// Mitsubishi GX Works2 project: Tap2V2FX3U   PLC: FX3U/FX3UC

// global labels: Global1
VAR_GLOBAL
  XXLimitN AT M8344 : BOOL;
  XXLimitP AT M8343 : BOOL;
  XXBusy AT M8340 : BOOL;
  XXInterruptInverse AT M8347 : BOOL;
  XXPos AT D8340 : DINT;
  XXAccelTime AT D8348 : INT;
  XXDecelTime AT D8349 : INT;
  XXPosView AT D0 : DINT;
  XXTarPos AT D2 : DINT;
  XXFeed AT D4 : DINT;
  XXPPR AT D6 : DINT;
  XXTarR AT M0 : BOOL;
  XXTarRSkip AT D8 : INT;
  XXOn AT M1 : BOOL;
  XXRun AT M2 : BOOL;
  XXDirection AT M3 : BOOL;
  XXMinI AT X000 : BOOL;
  XXReady AT M4 : BOOL;
  XXReadyI AT X004 : BOOL;
  XXPulseO AT Y000 : BOOL;
  XXDirectionO AT Y004 : BOOL;
  XXOnO AT Y010 : BOOL;
  XXInTorqueI AT X010 : BOOL;
  XXInTorqueIEdge AT M5 : BOOL;
  XXOverTorque AT M6 : BOOL;
  YYLimitN AT M8354 : BOOL;
  YYLimitP AT M8353 : BOOL;
  YYBusy AT M8350 : BOOL;
  YYInterruptInverse AT M8357 : BOOL;
  YYPos AT D8350 : DINT;
  YYAccelTime AT D8358 : INT;
  YYDecelTime AT D8359 : INT;
  YYPosView AT D9 : DINT;
  YYTarPos AT D11 : DINT;
  YYFeed AT D13 : DINT;
  YYPPM AT D15 : DINT;
  YYTarR AT M7 : BOOL;
  YYTarRSkip AT D17 : INT;
  YYOn AT M8 : BOOL;
  YYRun AT M9 : BOOL;
  YYDirection AT M10 : BOOL;
  YYReady AT M11 : BOOL;
  YYReadyI AT X005 : BOOL;
  YYPulseO AT Y001 : BOOL;
  YYDirectionO AT Y005 : BOOL;
  YYOnO AT Y011 : BOOL;
  YYInTorqueI AT X011 : BOOL;
  YYInTorqueIEdge AT M12 : BOOL;
  YYOverTorque AT M13 : BOOL;
  ZZLimitN AT M8364 : BOOL;
  ZZLimitP AT M8363 : BOOL;
  ZZBusy AT M8360 : BOOL;
  ZZInterruptInverse AT M8367 : BOOL;
  ZZPos AT D8360 : DINT;
  ZZAccelTime AT D8368 : INT;
  ZZDecelTime AT D8369 : INT;
  ZZPosView AT D18 : DINT;
  ZZTarPos AT D20 : DINT;
  ZZFeed AT D22 : DINT;
  ZZPPR AT D24 : DINT;
  ZZTarR AT M14 : BOOL;
  ZZTarRSkip AT D26 : INT;
  ZZRun AT M15 : BOOL;
  ZZDirection AT M16 : BOOL;
  ZZReadyI AT X006 : BOOL;
  ZZPulseO AT Y002 : BOOL;
  ZZDirectionO AT Y006 : BOOL;
  ZZOnO AT Y012 : BOOL;
  ZZInTorqueI AT X012 : BOOL;
  ZZInTorqueIEdge AT M17 : BOOL;
  ZZOverTorque AT M18 : BOOL;
  RunState AT D27 : INT;
  RunStateNext AT M19 : BOOL;
  AxisSpinState AT D28 : INT;
  AxisSpinStateNext AT M20 : BOOL;
  AxisTapState AT D29 : INT;
  AxisTapStateNext AT M21 : BOOL;
  FoilExtractState AT D30 : INT;
  FoilExtractStateNext AT M22 : BOOL;
  FoilClampState AT D31 : INT;
  FoilClampStateNext AT M23 : BOOL;
  FoilSupplyState AT D32 : INT;
  FoilSupplyStateNext AT M24 : BOOL;
  FoilExtractDropN AT M25 : BOOL;
  FoilExtractDropNTimer AT TC0 : BOOL;
  FoilExtractDropNTimerDelay AT D33 : INT;
  FoilExtractDropP AT M26 : BOOL;
  FoilExtractDropPTimer AT TC1 : BOOL;
  FoilExtractDropPTimerDelay AT D34 : INT;
  FoilExtractDrop AT M27 : BOOL;
  FoilExtractDropO AT Y003 : BOOL;
  FoilClampN AT M28 : BOOL;
  FoilClampNTimer AT TC2 : BOOL;
  FoilClampNTimerDelay AT D35 : INT;
  FoilClampP AT M29 : BOOL;
  FoilClampPTimer AT TC3 : BOOL;
  FoilClampPTimerDelay AT D36 : INT;
  FoilClampPI AT X001 : BOOL;
  FoilClamp AT M30 : BOOL;
  FoilClampO AT Y007 : BOOL;
  FoilSupply AT M31 : BOOL;
  FoilSupplyO AT Y013 : BOOL;
  WorkFeedSpin AT D37 : DINT;
  WorkFeedTapTravelFast AT D39 : DINT;
  WorkFeedTapSpinDown AT D41 : DINT;
  WorkFeedTapSpinUp AT D43 : DINT;
  FoilFull AT M32 : BOOL;
  FoilFullI AT X002 : BOOL;
  FoilFullTimer AT TC4 : BOOL;
  SpinArray AT D45 : ARRAY [0..7] OF DINT;
  SpinArrayIndex AT D61 : INT;
  AirReady AT M33 : BOOL;
  AirReadyI AT X003 : BOOL;
  Run AT M34 : BOOL;
  RunI AT X007 : BOOL;
  RunStop AT M35 : BOOL;
  RunStopI AT X013 : BOOL;
  SettingTapPitch AT D62 : DINT;
  SettingTapPitchI AT X014 : BOOL;
  SettingFoilSupplyI AT X015 : BOOL;
  SettingTapSpinSpeedI AT X016 : BOOL;
  SettingTapTravelLengthIObsolete AT X017 : BOOL;
  SettingTapTravelBegin AT D64 : DINT;
  SettingTapTravelBeginOffset AT D66 : DINT;
  SettingTapTravelFast AT D68 : DINT;
  SettingTapTravelEnd AT D70 : DINT;
  TapMoveToTravelBegin AT M36 : BOOL;
  TapCount AT D72 : DINT;
  TapCountAtSupplyEnd AT D74 : DINT;
  TapCountResetOrigin AT D76 : DINT;
  StopTap AT M37 : BOOL;
  StopTapTimer AT TC5 : BOOL;
  StopClamp AT M38 : BOOL;
  StopClampPLS AT M39 : BOOL;
  StopClampTimer AT TC6 : BOOL;
  XXOff AT M40 : BOOL;
  XXOffTimer AT TC7 : BOOL;
  Alert AT M41 : BOOL;
  AlertTimer AT TC8 : BOOL;
  AlertO AT Y014 : BOOL;
  ErrorReset AT M42 : BOOL;
  ErrorResetTimer AT TC9 : BOOL;
  ErrorResetO AT Y015 : BOOL;
  OverloadTimer AT TC256 : BOOL;
  OverloadTimerEN AT M43 : BOOL;
  Overload AT M44 : BOOL;
  SettingTapPitchBoolCounter1000 AT D78 : INT;
  SettingTapPitchBoolCounter1270 AT D79 : INT;
  SettingTapPitchBool AT M45 : BOOL;
  SettingTapPitchBoolO AT Y016 : BOOL;
  SettingTapPitchDone AT M46 : BOOL;
END_VAR

// task Task_01 (event TRUE, interval 0, priority 31): POU_01

PROGRAM POU_01
VAR
  fTmp : BOOL;
  fSpace : DINT;
  fCount : INT;
  fNeedResetOrigin : BOOL;
END_VAR
SET(M8002, M8336);
MOV(M8002, HFFF0, D8336);
RST(M8002, XXInterruptInverse);
RST(M8002, XXOn);
RST(M8002, YYOn);
MOV(M8002, 50, XXAccelTime);
MOV(M8002, 50, XXDecelTime);
MOV(M8002, 250, YYAccelTime); MOV(M8002, YYAccelTime, ZZAccelTime);
MOV(M8002, 250, YYDecelTime); MOV(M8002, YYDecelTime, ZZDecelTime);
RST(M8002, XXOverTorque);
RST(M8002, YYOverTorque);
RST(M8002, ZZOverTorque);
RST(M8002, FoilExtractDrop);
RST(M8002, FoilClamp);
RST(M8002, FoilSupply);
SET(M8002, Alert);
(*x axis: index spin*)
DMOV(M8002, 131_072, XXPPR);
MOV(M8002, 8, fCount);
DMOV(M8002, XXPPR / INT_TO_DINT(fCount), fSpace);
DMOV(M8002, fSpace * 0, SpinArray[0]);
DMOV(M8002, fSpace * 1, SpinArray[1]);
DMOV(M8002, fSpace * 2, SpinArray[2]);
DMOV(M8002, fSpace * 3, SpinArray[3]);
DMOV(M8002, fSpace * 4, SpinArray[4]);
DMOV(M8002, fSpace * 5, SpinArray[5]);
DMOV(M8002, fSpace * 6, SpinArray[6]);
DMOV(M8002, fSpace * 7, SpinArray[7]);
DMOV(M8002, 98_304, WorkFeedSpin);
(*y axis: tap travel*)
DMOV(M8002, 1_000, YYPPM);
RST(M8002, TapCount);
DMOV(M8002, 100_000, WorkFeedTapTravelFast);
(*z axis: tap spin*)
DMOV(M8002, YYPPM, ZZPPR);
(*it easier to calculate if YYPPM = ZZPPR*)
(*|||||||||||||||*)

(*|||||||||||||||*)
SET(Run AND RunState = 0 AND AirReady AND SettingTapPitchDone, fTmp);
RST(fTmp, Run);
SET(fTmp, XXOn);
SET(fTmp, YYOn);
SET(fTmp, TapMoveToTravelBegin);
RST(fTmp, StopClamp);
MOV(fTmp, 1, RunState);
RST(fTmp, fTmp);
SET(RunStop OR Overload, fTmp);
SET(fTmp AND RunStop, ErrorReset);
RST(fTmp, Run);
RST(fTmp, RunStop);
RST(fTmp, Overload);
SET(fTmp, Alert);
ZRST(fTmp, RunState, FoilSupplyState);
RST(fTmp, XXRun);
RST(fTmp, XXOn);
RST(fTmp, YYRun);
RST(fTmp, ZZRun);
SET(fTmp AND YYOn, StopTap);
RST(fTmp, FoilExtractDrop);
RST(fTmp, FoilClamp);
RST(fTmp, FoilSupply);
RST(fTmp, fTmp);
OUT_T(StopTap, StopTapTimer, 5);
RST(StopTapTimer, YYOn);
RST(StopTapTimer, StopTap);

(*|||||||||||||||*)
(*|||||||||||||||*)
INC(RunStateNext, RunState);
INC(AxisSpinStateNext, AxisSpinState);
INC(AxisTapStateNext, AxisTapState);
INC(FoilExtractStateNext, FoilExtractState);
INC(FoilClampStateNext, FoilClampState);
INC(FoilSupplyStateNext, FoilSupplyState);
ZRST(M8000, RunStateNext, FoilSupplyStateNext);
DECO(M8000, RunState, 6, M100);
DECO(M8000, AxisSpinState, 6, M200); DECO(M8000, AxisSpinState, 6, M1200); ZRST(NOT XXReady, M1200, M1263);
DECO(M8000, AxisTapState, 6, M300); DECO(M8000, AxisTapState, 6, M1300); ZRST(NOT YYReady, M1300, M1363);
DECO(M8000, FoilExtractState, 6, M400);
DECO(M8000, FoilClampState, 6, M500);
DECO(M8000, FoilSupplyState, 6, M600);
(*|||||||||||||||*)

(*|||||||||||||||*)
(*origin tap, extract, clamp, supply*)
MOV(M101, 1, AxisTapState);
MOV(M101, 1, FoilExtractState);
MOV(M101, 1, FoilClampState);
MOV(M101, 1, FoilSupplyState);
DMOV(M101, TapCount - 4, TapCountAtSupplyEnd);
DMOV(M101, TapCount + 30, TapCountResetOrigin);
SET(M101, RunStateNext);
(*origin spin*)
MOV(M102 AND M1320, 1, AxisSpinState);
SET(M102 AND M1320, RunStateNext);
(*ready done, run command -> cycle start*)
SET(M103 AND M1220 AND M1320 AND M420 AND M520 AND Run, RunStateNext);
(*cycle start*)
SET(M104 AND M1220 AND M1320 AND M420 AND M520, fTmp);
(**)
OUT(fTmp AND TapCount = TapCountResetOrigin, fNeedResetOrigin);
MOV(fNeedResetOrigin, 1, AxisTapState);
DMOV(fNeedResetOrigin, TapCount + 30, TapCountResetOrigin);
RST(fNeedResetOrigin, TapMoveToTravelBegin);
RST(fNeedResetOrigin, fTmp);
(**)
SET(fTmp, RunStateNext);
SET(fTmp, Alert);
RST(fTmp, fTmp);
(*clamp on*)
MOV(M105, 11, FoilClampState);
SET(M105, XXOff);
SET(M105, RunStateNext);
(*clamp on done -> tap, extract*)
SET(M106 AND M515, fTmp);
MOV(fTmp AND NOT XXOverTorque, 11, AxisTapState);
MOV(fTmp AND NOT XXOverTorque, 11, FoilExtractState);
MOV(fTmp, 11, RunState);
RST(fTmp, fTmp);
(*/////*)
(*/////*)
(*/////*)
(*tap done -> add tap count, clamp off*)
SET(M111 AND M1320, fTmp);
DINC(fTmp AND NOT XXOverTorque, TapCount);
MOV(fTmp, 16, FoilClampState);
SET(fTmp, RunStateNext);
RST(fTmp, fTmp);
(*clamp off done, extract drop done -> vibrate*)
SET(M112 AND M520 AND M420, fTmp);
SET(fTmp, XXOn);
MOV(fTmp, 16, AxisSpinState);
SET(fTmp, RunStateNext);
RST(fTmp, fTmp);
(*vibrate done -> next hole*)
SET(M113 AND M1220, fTmp);
RST(fTmp, XXOverTorque);
MOV(fTmp, 11, AxisSpinState);
MOV(fTmp, 31, RunState);
RST(fTmp, fTmp);
(*/////*)
(*/////*)
(*/////*)
(*next hole done -> reclamp || return cycle start*)
SET(M131 AND M1215, fTmp);
MOV(fTmp AND XXOverTorque, 5, RunState);
MOV(fTmp AND NOT XXOverTorque, 4, RunState);
RST(fTmp AND NOT XXOverTorque, Alert);
MOV(fTmp, 20, AxisSpinState);
RST(fTmp, fTmp);
(*|||||||||||||||*)
(*foil full -> record*)
DMOV(FoilFull, TapCount, TapCountAtSupplyEnd);
(*check*)
SET((TapCount - TapCountAtSupplyEnd) >= 4, fTmp);
RST(NOT SettingFoilSupplyI, fTmp);
OUT(fTmp AND NOT FoilFull AND M620, FoilSupply);
RST(fTmp, fTmp);
(*|||||||||||||||*)

(*|||||||||||||||*)
(*/////get origin spin*)
(*dvit(EN, offset, frequency)*)
DDVIT(M201, 16_384, 32_768, XXPulseO, XXDirection);
SET(M201 AND M8029, AxisSpinStateNext);
RST(M201 AND M8029, M201);
(*reset index and position*)
RST(M1202, SpinArrayIndex);
DMOV(M1202, -fSpace, XXPos);
MOV(M1202, 20, AxisSpinState);
(*reset index and position*)
RST(M1206, SpinArrayIndex);
DMOV(M1206, -fSpace, XXPos);
MOV(M1206, 12, AxisSpinState);
(*/////main sequence*)
(*re get origin or next*)
SET(M1211 AND SpinArrayIndex >= fCount, fTmp);
MOV(M1211 AND fTmp, 6, AxisSpinState);
SET(M1211 AND NOT fTmp, AxisSpinStateNext);
RST(fTmp, fTmp);
(*move to hole*)
DMOV(M1212, SpinArray[SpinArrayIndex], XXTarPos);
DMOV(M1212, WorkFeedSpin, XXFeed);
INC(M1212, SpinArrayIndex);
SET(M1212, XXRun);
MOV(M1212, 15, AxisSpinState);
(*/////vibrate sequence*)
(*back*)
DMOV(M1216, XXPos - 1024, XXTarPos);
DMOV(M1216, WorkFeedSpin, XXFeed);
SET(M1216, XXRun);
SET(M1216, AxisSpinStateNext);
(*forward*)
DMOV(M1217, XXPos + 1024, XXTarPos);
DMOV(M1217, WorkFeedSpin, XXFeed);
SET(M1217, XXRun);
SET(M1217, AxisSpinStateNext);
(*forward done -> end*)
MOV(M1218, 20, AxisSpinState);
(*|||||||||||||||*)


(*|||||||||||||||*)
(*/////get origin tap*)
(*move back*)
SET(M1301, fTmp);
RST(fTmp, YYPos); RST(fTmp, ZZPos);
DMOV(fTmp, -100_000, YYTarPos); DMOV(fTmp, YYTarPos * ZZPPR / SettingTapPitch, ZZTarPos);
DMOV(fTmp, 5_000, YYFeed); DMOV(fTmp, YYFeed * ZZPPR / SettingTapPitch, ZZFeed);
SET(fTmp, YYRun); SET(fTmp, ZZRun);
SET(fTmp, AxisTapStateNext);
RST(fTmp, fTmp);
(*move back hit hard limit -> reset*)
SET(M302 AND NOT YYBusy, fTmp);
RST(fTmp, YYRun); RST(fTmp, ZZRun);
RST(fTmp, YYPos); RST(fTmp, ZZPos);
SET(fTmp, AxisTapStateNext);
RST(fTmp, fTmp);
(*move forward*)
SET(M1303, fTmp);
DMOV(fTmp, 5_000, YYTarPos);
DMOV(fTmp, 1_000, YYFeed);
SET(fTmp, YYRun);
SET(fTmp, AxisTapStateNext);
RST(fTmp, fTmp);
(*move forward out hard limit -> stop*)
SET(M304 AND YYInTorqueI, fTmp);
RST(fTmp, YYRun);
SET(fTmp, AxisTapStateNext);
RST(fTmp, fTmp);
(*stop done -> move forward x mm*)
SET(M1305, fTmp);
DMOV(fTmp, YYPos + 1_000, YYTarPos);
DMOV(fTmp, 5_000, YYFeed);
SET(fTmp, YYRun);
SET(fTmp, AxisTapStateNext);
RST(fTmp, fTmp);
(*move forward x mm done -> reset, move to begin or end*)
SET(M1306, fTmp);
RST(fTmp, YYPos); RST(fTmp, ZZPos);
MOV(fTmp AND TapMoveToTravelBegin, 7, AxisTapState);
MOV(fTmp AND NOT TapMoveToTravelBegin, 8, AxisTapState);
RST(fTmp, fTmp);
(*move to begin*)
DMOV(M1307, SettingTapTravelBegin, YYTarPos);
DMOV(M1307, 20_000, YYFeed);
SET(M1307, YYRun);
SET(M1307, AxisTapStateNext);
(*ready*)
MOV(M1308, 20, AxisTapState);
(*/////main sequence*)
(*move forward fast*)
SET(M1311, fTmp);
DMOV(fTmp, SettingTapTravelFast, YYTarPos);
DMOV(fTmp, WorkFeedTapTravelFast, YYFeed);
SET(fTmp, YYRun);
SET(fTmp, AxisTapStateNext); RST(fTmp, fTmp);
(*move forward fast done -> move forward*)
SET(M1312, fTmp);
DMOV(fTmp, SettingTapTravelEnd, YYTarPos); RST(fTmp, ZZPos); DMOV(fTmp, (YYTarPos - YYPos) * ZZPPR / SettingTapPitch, ZZTarPos);
DMOV(fTmp, WorkFeedTapSpinDown, ZZFeed); DMOV(fTmp, ZZFeed * SettingTapPitch / ZZPPR, YYFeed);
SET(fTmp, YYRun); SET(fTmp, ZZRun);
SET(fTmp, AxisTapStateNext); RST(fTmp, fTmp);
(*move forward done -> backlash eliminate*)
SET(M1313, fTmp);
DMOV(fTmp, ZZPos + 0_000, ZZTarPos);
DMOV(fTmp, 10_000, ZZFeed);
SET(fTmp, ZZRun);
SET(fTmp, AxisTapStateNext); RST(fTmp, fTmp);
(*backlash eliminate done -> move back*)
SET(M1314, fTmp);
DMOV(fTmp, SettingTapTravelBegin + SettingTapTravelBeginOffset, YYTarPos); RST(fTmp, ZZPos); DMOV(fTmp, (YYTarPos - YYPos) * ZZPPR / SettingTapPitch, ZZTarPos);
DMOV(fTmp, WorkFeedTapSpinUp, ZZFeed); DMOV(fTmp, ZZFeed * SettingTapPitch / ZZPPR, YYFeed);
SET(fTmp, YYRun); SET(fTmp, ZZRun);
SET(fTmp, AxisTapStateNext); RST(fTmp, fTmp);
(*move back done -> end*)
SET(M1315, fTmp);
MOV(fTmp, 20, AxisTapState); RST(fTmp, fTmp);
(*|||||||||||||||*)

(*|||||||||||||||*)
(*/////get origin foil extract*)
(*drop back*)
RST(M401, FoilExtractDrop);
SET(M401, FoilExtractStateNext);
(*drop back done -> next*)
SET(M402 AND FoilExtractDropN, FoilExtractStateNext);
(*end*)
MOV(M403, 20, FoilExtractState);
(*/////drop sequence*)
(*drop forward*)
SET(M411, FoilExtractDrop);
SET(M411, FoilExtractStateNext);
(*drop forward done -> drop back*)
RST(M412 AND FoilExtractDropP, FoilExtractDrop);
SET(M412 AND FoilExtractDropP, FoilExtractStateNext);
(*drop back done -> end*)
MOV(M413 AND FoilExtractDropN, 20, FoilExtractState);
(*|||||||||||||||*)

(*|||||||||||||||*)
(*/////get origin foil clamp*)
(*back*)
RST(M501, FoilClamp);
SET(M501, FoilClampStateNext);
(*back done -> next*)
SET(M502 AND FoilClampN, FoilClampStateNext);
(*end*)
MOV(M503, 20, FoilClampState);
(*/////clamp on*)
(*forward*)
SET(M511, FoilClamp);
SET(M511, FoilClampStateNext);
(*forward done -> done*)
MOV(M512 AND FoilClampP, 15, FoilClampState);
(*/////clamp off*)
(*back*)
RST(M516, FoilClamp);
SET(M516, FoilClampStateNext);
(*back done -> done*)
MOV(M517 AND FoilClampN, 20, FoilClampState);
(*|||||||||||||||*)

(*|||||||||||||||*)
(*/////get origin foil supply*)
(*reset*)
RST(M601, FoilSupply);
SET(M601, FoilSupplyStateNext);
(*end*)
MOV(M602, 20, FoilSupplyState);
(*/////supply sequence*)
(*|||||||||||||||*)

(*|||||||||||||||*)
(*XX*)
RST(XXRun AND XXTarPos = XXPos, XXRun);
DDRVA(XXRun, XXTarPos, XXFeed, XXPulseO, XXDirection);
RST(M8029, XXRun);
OUT(XXDirection, XXDirectionO);
INC(NOT XXRun AND NOT XXBusy AND XXTarRSkip < 5, XXTarRSkip);
RST(XXRun, XXTarRSkip);
OUT(XXTarRSkip >= 5, XXTarR);
(*|||||||||||||||*)
(*YY*)
RST(YYRun AND YYTarPos = YYPos, YYRun);
DDRVA(YYRun, YYTarPos, YYFeed, YYPulseO, YYDirection);
RST(M8029, YYRun);
OUT(NOT YYDirection, YYDirectionO);
INC(NOT YYRun AND NOT YYBusy AND YYTarRSkip < 5, YYTarRSkip);
RST(YYRun, YYTarRSkip);
OUT(YYTarRSkip >= 5, YYTarR);
(*|||||||||||||||*)
(*ZZ*)
RST(ZZRun AND ZZTarPos = ZZPos, ZZRun);
DDRVA(ZZRun, ZZTarPos, ZZFeed, ZZPulseO, ZZDirection);
RST(M8029, ZZRun);
OUT(NOT ZZDirection, ZZDirectionO);
INC(NOT ZZRun AND NOT ZZBusy AND ZZTarRSkip < 5, ZZTarRSkip);
RST(ZZRun, ZZTarRSkip);
OUT(ZZTarRSkip >= 5, ZZTarR);
(*|||||||||||||||*)
(*ready*)
OUT(XXReadyI AND XXTarR, XXReady);
OUT(YYReadyI AND YYTarR AND ZZReadyI AND ZZTarR, YYReady);
(*limit*)
OUT(NOT YYDirection AND NOT YYInTorqueI AND AxisTapState <= 10, YYLimitN); OUT(YYLimitN, ZZLimitN);
(*|||||||||||||||*)

(*|||||||||||||||*)
PLS(RunI, Run); SET(Run, Run);
PLF(RunStopI, RunStop); SET(RunStop, RunStop);
OUT_T(NOT RunStopI AND NOT StopClamp, StopClampTimer, 20); SET(StopClampTimer, StopClamp);
RST(StopClamp, RunStop);
SET(StopClamp, FoilClamp);
SET(StopClamp AND FoilClampP, fTmp);
SET(fTmp, YYOn);
MOV(fTmp, 1, AxisTapState);
RST(fTmp, StopClamp);
RST(fTmp, TapMoveToTravelBegin);
RST(fTmp, fTmp);
PLF(XXInTorqueI, XXInTorqueIEdge); SET(XXInTorqueIEdge AND NOT XXOff, XXOverTorque);
OUT(NOT YYInTorqueI AND AxisTapState > 10, OverloadTimerEN); OUT_T(OverloadTimerEN, OverloadTimer, 50); SET(OverloadTimer, Overload);
(*foil extract*)
MOV(M8002, 2, FoilExtractDropNTimerDelay);
OUT_T(NOT FoilExtractDrop, FoilExtractDropNTimer, FoilExtractDropNTimerDelay); SET(FoilExtractDropNTimer, FoilExtractDropN); RST(FoilExtractDropNTimer, FoilExtractDropP);
MOV(M8002, 5, FoilExtractDropPTimerDelay);
OUT_T(FoilExtractDrop, FoilExtractDropPTimer, FoilExtractDropPTimerDelay); SET(FoilExtractDropPTimer, FoilExtractDropP); RST(FoilExtractDropPTimer, FoilExtractDropN);
(*foil clamp*)
MOV(M8002, 3, FoilClampNTimerDelay);
OUT_T(NOT FoilClamp AND NOT FoilClampPI, FoilClampNTimer, FoilClampNTimerDelay); SET(FoilClampNTimer, FoilClampN); RST(FoilClampNTimer, FoilClampP);
MOV(M8002, 1, FoilClampPTimerDelay);
OUT_T(FoilClamp AND FoilClampPI, FoilClampPTimer, FoilClampPTimerDelay); SET(FoilClampPTimer, FoilClampP); RST(FoilClampPTimer, FoilClampN);
(*foil supply*)
OUT_T(FoilFullI, FoilFullTimer, 5); OUT(FoilFullTimer, FoilFull);
(*setting pitch*)
RST(M8002, SettingTapPitchDone);
RST(M8002, SettingTapPitchBoolCounter1000);
RST(M8002, SettingTapPitchBoolCounter1270);
INC(M8000 AND NOT SettingTapPitchDone AND NOT SettingTapPitchI, SettingTapPitchBoolCounter1000);
INC(M8000 AND NOT SettingTapPitchDone AND SettingTapPitchI, SettingTapPitchBoolCounter1270);
SET(SettingTapPitchBoolCounter1000 > 500 OR SettingTapPitchBoolCounter1270 > 500, fTmp);
RST(fTmp AND SettingTapPitchBoolCounter1000 > SettingTapPitchBoolCounter1270, SettingTapPitchBool);
SET(fTmp AND SettingTapPitchBoolCounter1270 > SettingTapPitchBoolCounter1000, SettingTapPitchBool);
DMOV(fTmp AND NOT SettingTapPitchBool, 1_000, SettingTapPitch);
DMOV(fTmp AND SettingTapPitchBool, 1_270, SettingTapPitch);
SET(fTmp, SettingTapPitchDone);
RST(fTmp, fTmp);
OUT(SettingTapPitchBool, SettingTapPitchBoolO);
(*setting feed*)
(*M6*)
DMOV(NOT SettingTapPitchBool AND NOT SettingTapSpinSpeedI, (ZZPPR * 1_400) / 60, WorkFeedTapSpinDown);
DMOV(NOT SettingTapPitchBool AND NOT SettingTapSpinSpeedI, (ZZPPR * 1_400) / 60, WorkFeedTapSpinUp);
DMOV(NOT SettingTapPitchBool AND SettingTapSpinSpeedI, (ZZPPR * 1_600) / 60, WorkFeedTapSpinDown);
DMOV(NOT SettingTapPitchBool AND SettingTapSpinSpeedI, (ZZPPR * 1_600) / 60, WorkFeedTapSpinUp);
(*1/4*)
DMOV(SettingTapPitchBool AND NOT SettingTapSpinSpeedI, (ZZPPR * 1_200) / 60, WorkFeedTapSpinDown);
DMOV(SettingTapPitchBool AND NOT SettingTapSpinSpeedI, (ZZPPR * 1_200) / 60, WorkFeedTapSpinUp);
DMOV(SettingTapPitchBool AND SettingTapSpinSpeedI, (ZZPPR * 1_400) / 60, WorkFeedTapSpinDown);
DMOV(SettingTapPitchBool AND SettingTapSpinSpeedI, (ZZPPR * 1_400) / 60, WorkFeedTapSpinUp);
(*setting travel*)
DMOV(M8002, 10_000, SettingTapTravelBegin);
DMOV(M8002, SettingTapTravelBegin + 25_000, SettingTapTravelEnd);
DMOV(M8002, SettingTapTravelBegin + 1_000, SettingTapTravelFast);
DMOV(M8002, 0_000, SettingTapTravelBeginOffset);
(**)
OUT(AirReadyI, AirReady);
(*|||||||||||||||*)
OUT(XXOn, XXOnO);
OUT(YYOn, YYOnO); OUT(YYOn, ZZOnO);
OUT(FoilExtractDrop, FoilExtractDropO);
OUT(FoilClamp, FoilClampO);
OUT(FoilSupply, FoilSupplyO);
OUT(AlertTimer, AlertO);
OUT(ErrorReset, ErrorResetO);
(**)
OUT_T(XXOff, XXOffTimer, 5); RST(XXOffTimer, XXOn); RST(XXOffTimer, XXOff);
OUT_T(ErrorReset, ErrorResetTimer, 1); RST(ErrorResetTimer, ErrorReset);
RST(ErrorResetTimer, XXOverTorque);
RST(ErrorResetTimer, YYOverTorque);
RST(ErrorResetTimer, ZZOverTorque);
OUT_T(Alert, AlertTimer, 100);
(*|||||||||||||||*)
END_PROGRAM
